{attribute 'qualified_only'}
VAR_GLOBAL
	// Von Gewerk 2 zu Gewerk 3
	gvFahrvektor 	: sFahrvektor;
	gvZielPosition  : sPositions;
	inControl : RobotControl;     // Steuerungsvariable      // 0=idle, 1=Stop, 2=Reset, 3=Vektor, 4=Position
	
	// Von Gewerk 3 zu Gewerk 2
	gvActualPosition	: sPositions;
	inStatus			: RobotStatus; // Statusvariable	// 0=offline, 1=Betriebsbereit, 2=Laufend, 3=Ziel Erreicht, 4=Fehler
END_VAR

(* stored: Version 1.1.0.1, ProductVersion 3.1.4026.13
   GVL GVL_Datatransfer23: Id {5499bb5a-06ba-4b61-acc2-672869a8aa83} *)
